FUNCTION_BLOCK FB_Joint
VAR_INPUT
END_VAR
VAR_OUTPUT
END_VAR
VAR
	// motor IO
	m_motorInputs AT%I*	:ST_MotorInputs;
	m_motorOutputs AT%Q* :ST_MotorOutputs;
	
	// calibrated link encoder data
	m_minLinkEncoder :DINT;
	m_maxLinkEncoder :DINT;
	m_caliLinkEncoder :DINT;
	m_linkEncCaliJntPos :LREAL;
	m_linkEncZeroCross :INT;
	m_initMotorEnc : DINT;
	
	// joint position from link encoder after power on
	m_initLinkPos :LREAL;
	
	// data for link encoder multiple cycles
	m_lastLinkEncoder :DINT;
	m_linkEncCycles:INT;
	
	// device paramters
	m_motorEncoderRes :DINT;
	m_linkEncoderRes :DINT;
	m_motorReduction :LREAL;
	m_linkEncoderReduction :LREAL;
	m_trqConst :LREAL;
	m_maxCurrent :LREAL;
	m_motorDir :INT;								
	m_linkEncoderDir :INT;
	m_minJntPos: LREAL;
	m_maxJntPos: LREAL;
	
	// macro defined data for quick calculation
	m_trq2CurrentRatio:LREAL;
	m_current2TrqRatio:LREAL;
	m_linkEnc2PosRatio :LREAL;
	m_motorEnc2PosRatio :LREAL;
	
	// joint data
	m_curMotorPos :LREAL;
	m_curLinkPos :LREAL;
	m_curJntPos	:LREAL;
	m_curJntVel :LREAL;
	m_curJntTrq :	LREAL;
	m_cmdJntPos :LREAL;
	m_cmdJntVel :LREAL;
	m_cmdJntTrq :LREAL;
	m_lastJntPos :LREAL;
	
	// velocity filter
	m_jntVelLpf :FB_LowPassFilter;
	
	// command torque filter
	m_cmdTrqLpf :FB_LowPassFilter;
	
END_VAR

METHOD PUBLIC disable : BOOL
VAR_INPUT
END_VAR
m_motorOutputs.m_controlWord:=DriverCtrlWord_INIT;
disable:=true;
END_METHOD

METHOD PUBLIC enable : BOOL
VAR_INPUT
END_VAR
IF DriverStatusWord_INIT = m_motorInputs.m_statusWord THEN
	m_motorOutputs.m_controlWord:=DriverCtrlWord_PREOP;
	enable := FALSE;
ELSIF DriverStatusWord_PREOP = m_motorInputs.m_statusWord THEN
	m_motorOutputs.m_controlWord:=DriverCtrlWord_OP;
	enable :=  FALSE;
ELSIF DriverStatusWord_OP = m_motorInputs.m_statusWord THEN
	enable :=  TRUE;
//ELSE
//	m_motorOutputs.m_controlWord:=DriverCtrlWord_INIT;
//	enable :=  FALSE;
END_IF
END_METHOD

METHOD PUBLIC init : BOOL
VAR_INPUT
	i_armIdx :INT;
	i_jntIdx :INT;
END_VAR
// hardware parameters
m_motorEncoderRes :=g_incEncoderRes[i_jntIdx];
m_linkEncoderRes :=g_absEncoderRes[i_jntIdx];
m_motorReduction :=g_motorReduction[i_jntIdx];
m_linkEncoderReduction :=g_absEncoderReduction[i_jntIdx];
m_trqConst :=g_motorTrqConst[i_jntIdx];
m_maxCurrent :=g_motorMaxCurrent[i_jntIdx];
m_motorDir :=g_motorDir[i_armIdx,i_jntIdx];								
m_linkEncoderDir :=g_asbEncoderDir[i_armIdx,i_jntIdx];
m_minJntPos	:=g_minJntPos[i_armIdx,i_jntIdx];
m_maxJntPos	:=g_maxJntPos[i_armIdx,i_jntIdx];

//link encoder calibartion data
m_minLinkEncoder :=g_minLinkEncoder[i_armIdx, i_jntIdx];
m_maxLinkEncoder :=g_maxLinkEncoder[i_armIdx, i_jntIdx];
m_caliLinkEncoder :=g_caliLinkEncoder[i_armIdx, i_jntIdx];
m_linkEncCaliJntPos :=g_linkEncCaliJntPos[i_armIdx, i_jntIdx];
m_linkEncZeroCross :=g_linkEncZeroCross[i_armIdx, i_jntIdx];

// convert cali link encoder if joint cross zero
IF 1=m_linkEncZeroCross THEN
	IF 1=m_linkEncoderDir AND m_caliLinkEncoder < m_minLinkEncoder THEN
		m_caliLinkEncoder := g_caliLinkEncoder[i_armIdx, i_jntIdx] + m_linkEncoderRes;
	ELSIF -1=m_linkEncoderDir AND m_caliLinkEncoder < m_maxLinkEncoder THEN
		m_caliLinkEncoder := g_caliLinkEncoder[i_armIdx, i_jntIdx] + m_linkEncoderRes;
	END_IF
END_IF

// compute link and motor pos
//!NOTICE: Need to be reset after joint back to center for multiple cycle joints
m_lastLinkEncoder :=m_motorInputs.m_linkEncoder;
m_linkEncCycles:=0;
m_curLinkPos :=linkEnc2Pos();
m_initLinkPos:=m_curLinkPos;
m_initMotorEnc :=m_motorInputs.m_motorEncoder;
m_curMotorPos :=motorEnc2Pos();	

// macro data
m_trq2CurrentRatio:=m_motorDir * 1000.0/(m_trqConst*m_motorReduction);
m_current2TrqRatio:=m_motorDir * (m_trqConst*m_motorReduction)/1000.0;
m_linkEnc2PosRatio := 2*PI*m_linkEncoderDir/(m_linkEncoderReduction*m_linkEncoderRes);
m_motorEnc2PosRatio := 2*PI * m_motorDir/(m_motorReduction * m_motorEncoderRes);

// motor data init
m_curJntPos := m_curMotorPos;
m_curJntVel:=0;
m_curJntTrq :=0;
m_cmdJntPos :=m_curJntPos;
m_cmdJntVel :=0.0;
m_cmdJntTrq :=0.0;
m_lastJntPos :=m_curJntPos;
m_jntVelLpf.init(1, g_curJntVelLpfCutoffFreq, g_armControlFreq);
m_cmdTrqLpf.init(1, g_cmdJntTrqLpfCutoffFreq, g_armControlFreq);

// driver init value
m_motorOutputs.m_controlWord:=DriverCtrlWord_INIT;
m_motorOutputs.m_opMode:=INT_TO_SINT(DriverOPMode_Pos);
m_motorOutputs.m_cmdCurrent:=0;
m_motorOutputs.m_cmdMotorEncoder:=m_motorInputs.m_motorEncoder;
END_METHOD

METHOD isEnabled : BOOL
VAR_INPUT
END_VAR
isEnabled :=(DriverStatusWord_OP = m_motorInputs.m_statusWord);
END_METHOD

PROPERTY jntPos : LREAL
GET
jntPos := m_curJntPos;
END_GET
END_PROPERTY

PROPERTY jntTrq : LREAL
GET
jntTrq:=m_curJntTrq;
END_GET
END_PROPERTY

PROPERTY jntVel : LREAL
GET
jntVel := m_curJntVel;
END_GET
END_PROPERTY

METHOD PROTECTED linkEnc2Pos : LREAL
VAR_INPUT
END_VAR
VAR
	incLinkPos :LREAL;
	newLinkEnc :DINT;
END_VAR
// cycle check
IF (m_motorInputs.m_linkEncoder - m_lastLinkEncoder)*m_linkEncoderDir < -m_linkEncoderRes/2 THEN
	m_linkEncCycles :=m_linkEncCycles+1;
ELSIF (m_motorInputs.m_linkEncoder - m_lastLinkEncoder)*m_linkEncoderDir > m_linkEncoderRes/2 THEN
	m_linkEncCycles :=m_linkEncCycles-1;
END_IF
m_lastLinkEncoder:=m_motorInputs.m_linkEncoder;

// convert link encoder if joint cross zero
newLinkEnc := m_motorInputs.m_linkEncoder;
IF 1=m_linkEncZeroCross THEN
	IF 1=m_linkEncoderDir AND m_motorInputs.m_linkEncoder < m_minLinkEncoder THEN
		newLinkEnc := m_motorInputs.m_linkEncoder + m_linkEncoderRes;
	ELSIF -1=m_linkEncoderDir AND m_motorInputs.m_linkEncoder < m_maxLinkEncoder THEN
		newLinkEnc := m_motorInputs.m_linkEncoder + m_linkEncoderRes;
	END_IF
END_IF

// motion from calibrated points
incLinkPos := (newLinkEnc-m_caliLinkEncoder)*m_linkEnc2PosRatio;

// absolute joint position
linkEnc2Pos := incLinkPos + m_linkEncCaliJntPos + 2*PI* m_linkEncCycles;
END_METHOD

PROPERTY PUBLIC linkPos : LREAL
GET
linkPos:=m_curLinkPos;
END_GET
END_PROPERTY

METHOD PROTECTED motorEnc2Pos : LREAL
VAR_INPUT
END_VAR
motorEnc2Pos:= (m_motorInputs.m_motorEncoder-m_initMotorEnc)* m_motorEnc2PosRatio +m_initLinkPos;
END_METHOD

PROPERTY PUBLIC motorPos : LREAL
GET
motorPos := m_curMotorPos;
END_GET
END_PROPERTY

// TODO
METHOD PROTECTED motorPos2Enc : DINT
VAR_INPUT
	i_jntPos :LREAL;
END_VAR

VAR
END_VAR
motorPos2Enc := LREAL_TO_DINT((i_jntPos-m_initLinkPos)/m_motorEnc2PosRatio + m_initMotorEnc);
END_METHOD

METHOD resetEncoder : BOOL
VAR_INPUT
END_VAR
m_lastLinkEncoder :=m_motorInputs.m_linkEncoder;
m_linkEncCycles:=0;
m_initMotorEnc :=m_motorInputs.m_motorEncoder;
m_curLinkPos :=linkEnc2Pos();
m_curMotorPos :=motorEnc2Pos();	
m_initLinkPos:=m_curLinkPos;
END_METHOD

METHOD PUBLIC updateCmds : BOOL
VAR_INPUT
	i_opMode : E_DriverOPMode;
	i_cmdPos :LREAL;
	i_cmdTrq :LREAL;
END_VAR
m_motorOutputs.m_opMode:=INT_TO_SINT( i_opMode);
// pos mode
IF i_opMode = DriverOPMode_Pos THEN
	m_motorOutputs.m_cmdCurrent:=0;
	m_motorOutputs.m_cmdMotorEncoder :=motorPos2Enc(i_cmdPos);
ELSIF i_opMode = DriverOPMode_Trq THEN
	m_motorOutputs.m_cmdCurrent:=LREAL_TO_DINT(LIMIT(-m_maxCurrent, i_cmdTrq*m_trq2CurrentRatio,m_maxCurrent));
	m_motorOutputs.m_cmdMotorEncoder :=m_motorInputs.m_motorEncoder; 
END_IF
END_METHOD

METHOD PUBLIC updateStatus : BOOL
VAR_INPUT
END_VAR
// compute joint position
m_curLinkPos:= linkEnc2Pos();
m_curMotorPos:=motorEnc2Pos();
m_curJntPos := m_curMotorPos;

// compute joint velocity
m_curJntVel:= (m_curJntPos-m_lastJntPos)/g_armControlLoopInterval;
m_curJntVel := m_jntVelLpf.run(m_curJntVel);

m_curJntTrq := m_motorInputs.m_current * m_current2TrqRatio;
END_METHOD

END_FUNCTION_BLOCK

(* stored: Version 1.1.0.1, ProductVersion 3.1.4024.11
   POU FB_Joint: Id {9ce08388-a134-4497-8af1-f051329728ca}, SpecialFunc None
   Folder property: Id {cdcb62c8-2a8b-4700-ad38-db65527ef407}
   Method disable: Id {e31df8a7-8ce0-47c3-be01-feb458684c41}
   Method enable: Id {cf1e8549-8fbc-49c1-a41e-ead1f2db1255}
   Method init: Id {9b72c880-30e6-407f-a349-f349818eddee}
   Method isEnabled: Id {6575d317-fe99-4038-982b-c3651c898873}
   Property jntPos: Id {7c60c4ea-0665-427c-81ff-ecca027383e5}
   Get Get: Id {0999bfb4-2d73-48db-9f0b-eb60a7757215}
   Property jntTrq: Id {24f2edfa-7ea0-460c-b46c-37e80340999b}
   Get Get: Id {a73a2159-96f0-4307-8408-692459f39004}
   Property jntVel: Id {9f6c9647-33be-4e59-a761-fc40f97a604f}
   Get Get: Id {dda73f9b-c1f5-4fa7-a73f-7b4550e82f69}
   Method linkEnc2Pos: Id {ee202f01-7eae-4c96-9148-de033a227f8f}
   Property linkPos: Id {e503da77-c373-4ba2-b314-228646ff52c0}
   Get Get: Id {057e650e-064f-4e5d-ae71-67363977daff}
   Method motorEnc2Pos: Id {5111dbab-73a3-4041-b0b2-3d1b70394152}
   Property motorPos: Id {257e5d05-bbd2-45b4-a27c-60112e2ac416}
   Get Get: Id {5c2a1542-7420-4542-ba4a-8202be5bc4e5}
   Method motorPos2Enc: Id {5927a17d-d8e9-40fc-9c34-e6793775a7fc}
   Method resetEncoder: Id {c1110436-e250-45fb-8008-63b89ff1e4a3}
   Method updateCmds: Id {a4f5fe94-40e9-4f77-a4d8-a2af848a52e6}
   Method updateStatus: Id {77cc6f91-59d3-42a9-8d8a-2f8d584653fb} *)
